// Mitsubishi GX Works2 project: CODE_PLC_HMI   PLC: FX1N/FX1NC

PROGRAM MAIN
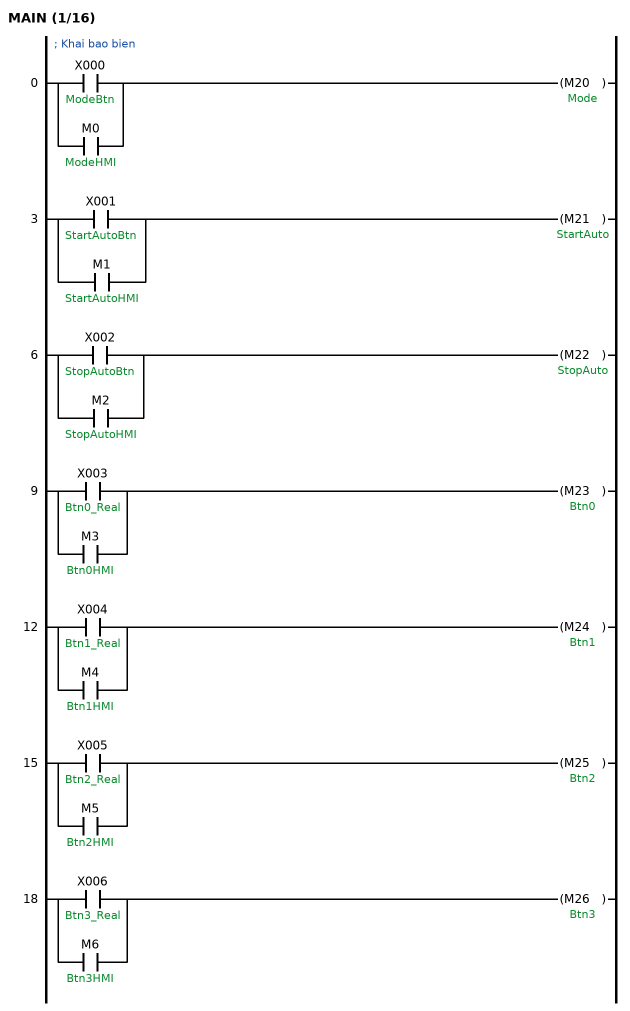
; Khai bao bien
0     LD      X000  ; ModeBtn
      OR      M0  ; ModeHMI
      OUT     M20  ; Mode
3     LD      X001  ; StartAutoBtn
      OR      M1  ; StartAutoHMI
      OUT     M21  ; StartAuto
6     LD      X002  ; StopAutoBtn
      OR      M2  ; StopAutoHMI
      OUT     M22  ; StopAuto
9     LD      X003  ; Btn0_Real
      OR      M3  ; Btn0HMI
      OUT     M23  ; Btn0
12    LD      X004  ; Btn1_Real
      OR      M4  ; Btn1HMI
      OUT     M24  ; Btn1
15    LD      X005  ; Btn2_Real
      OR      M5  ; Btn2HMI
      OUT     M25  ; Btn2
18    LD      X006  ; Btn3_Real
      OR      M6  ; Btn3HMI
      OUT     M26  ; Btn3
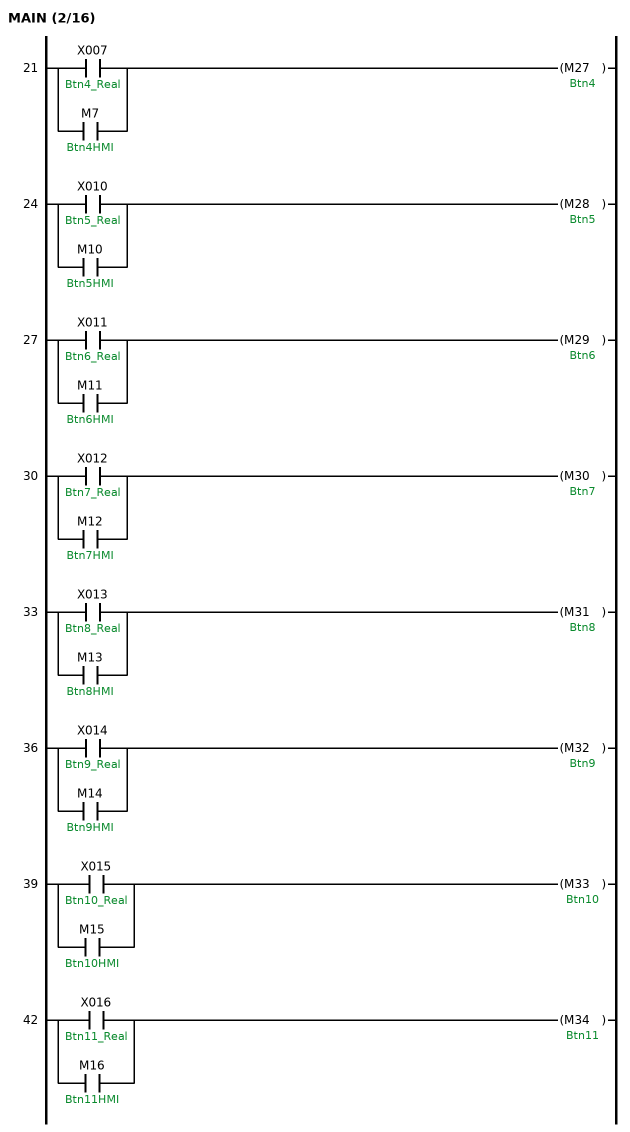
21    LD      X007  ; Btn4_Real
      OR      M7  ; Btn4HMI
      OUT     M27  ; Btn4
24    LD      X010  ; Btn5_Real
      OR      M10  ; Btn5HMI
      OUT     M28  ; Btn5
27    LD      X011  ; Btn6_Real
      OR      M11  ; Btn6HMI
      OUT     M29  ; Btn6
30    LD      X012  ; Btn7_Real
      OR      M12  ; Btn7HMI
      OUT     M30  ; Btn7
33    LD      X013  ; Btn8_Real
      OR      M13  ; Btn8HMI
      OUT     M31  ; Btn8
36    LD      X014  ; Btn9_Real
      OR      M14  ; Btn9HMI
      OUT     M32  ; Btn9
39    LD      X015  ; Btn10_Real
      OR      M15  ; Btn10HMI
      OUT     M33  ; Btn10
42    LD      X016  ; Btn11_Real
      OR      M16  ; Btn11HMI
      OUT     M34  ; Btn11
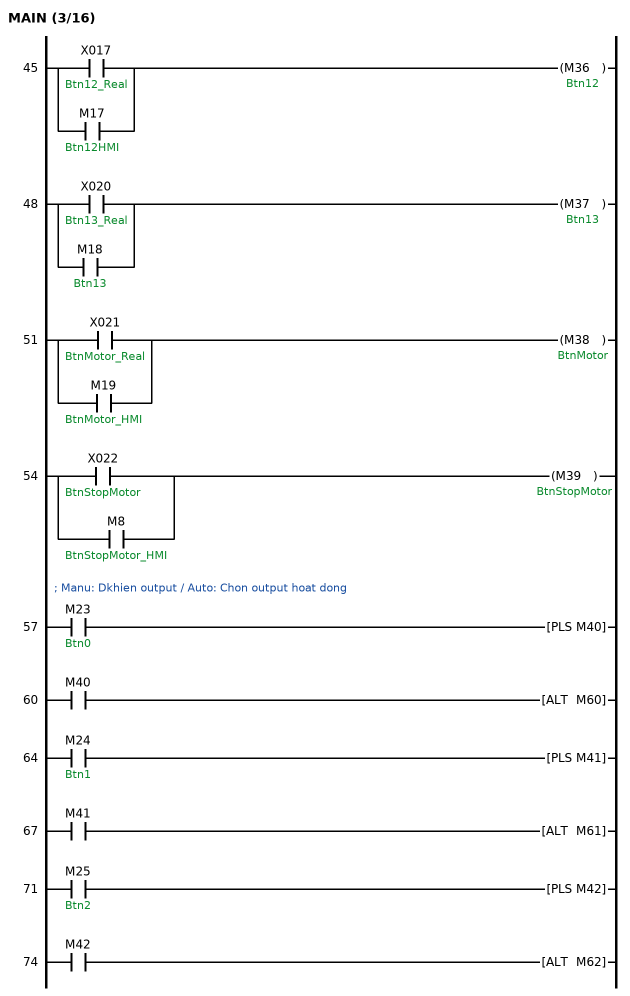
45    LD      X017  ; Btn12_Real
      OR      M17  ; Btn12HMI
      OUT     M36  ; Btn12
48    LD      X020  ; Btn13_Real
      OR      M18  ; Btn13
      OUT     M37  ; Btn13
51    LD      X021  ; BtnMotor_Real
      OR      M19  ; BtnMotor_HMI
      OUT     M38  ; BtnMotor
54    LD      X022  ; BtnStopMotor
      OR      M8  ; BtnStopMotor_HMI
      OUT     M39  ; BtnStopMotor
; Manu: Dkhien output / Auto: Chon output hoat dong
57    LD      M23  ; Btn0
      PLS     M40
60    LD      M40
      ALT     M60
64    LD      M24  ; Btn1
      PLS     M41
67    LD      M41
      ALT     M61
71    LD      M25  ; Btn2
      PLS     M42
74    LD      M42
      ALT     M62
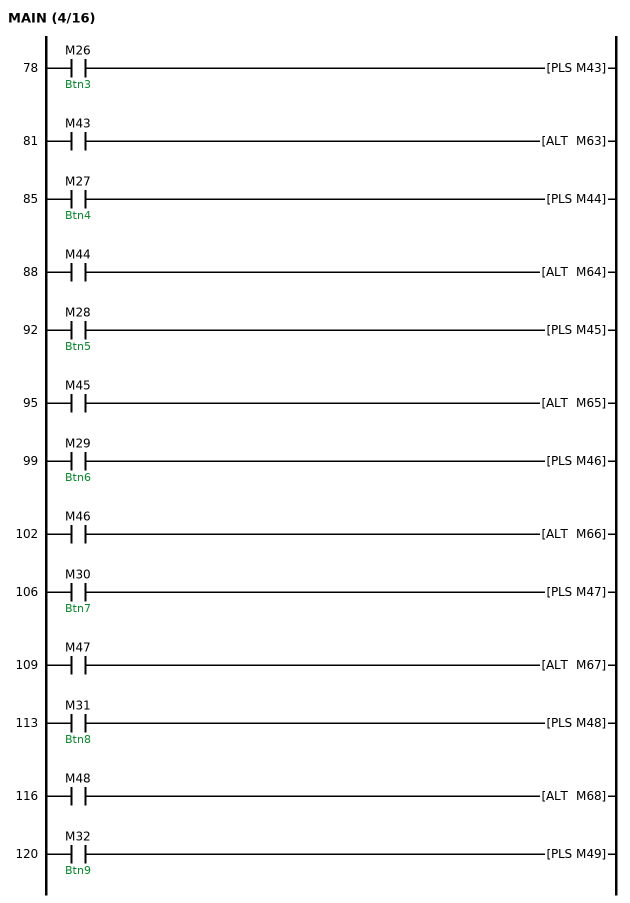
78    LD      M26  ; Btn3
      PLS     M43
81    LD      M43
      ALT     M63
85    LD      M27  ; Btn4
      PLS     M44
88    LD      M44
      ALT     M64
92    LD      M28  ; Btn5
      PLS     M45
95    LD      M45
      ALT     M65
99    LD      M29  ; Btn6
      PLS     M46
102   LD      M46
      ALT     M66
106   LD      M30  ; Btn7
      PLS     M47
109   LD      M47
      ALT     M67
113   LD      M31  ; Btn8
      PLS     M48
116   LD      M48
      ALT     M68
120   LD      M32  ; Btn9
      PLS     M49
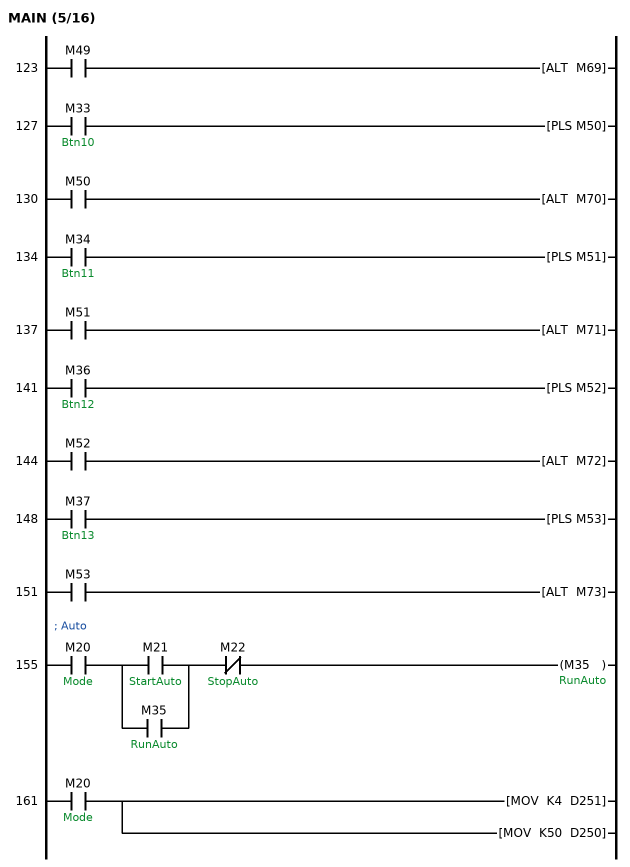
123   LD      M49
      ALT     M69
127   LD      M33  ; Btn10
      PLS     M50
130   LD      M50
      ALT     M70
134   LD      M34  ; Btn11
      PLS     M51
137   LD      M51
      ALT     M71
141   LD      M36  ; Btn12
      PLS     M52
144   LD      M52
      ALT     M72
148   LD      M37  ; Btn13
      PLS     M53
151   LD      M53
      ALT     M73
; 
; Auto
155   LD      M20  ; Mode
      LD      M21  ; StartAuto
      OR      M35  ; RunAuto
      ANB
      ANI     M22  ; StopAuto
      OUT     M35  ; RunAuto
161   LD      M20  ; Mode
      MOV     K4 D251
      MOV     K50 D250
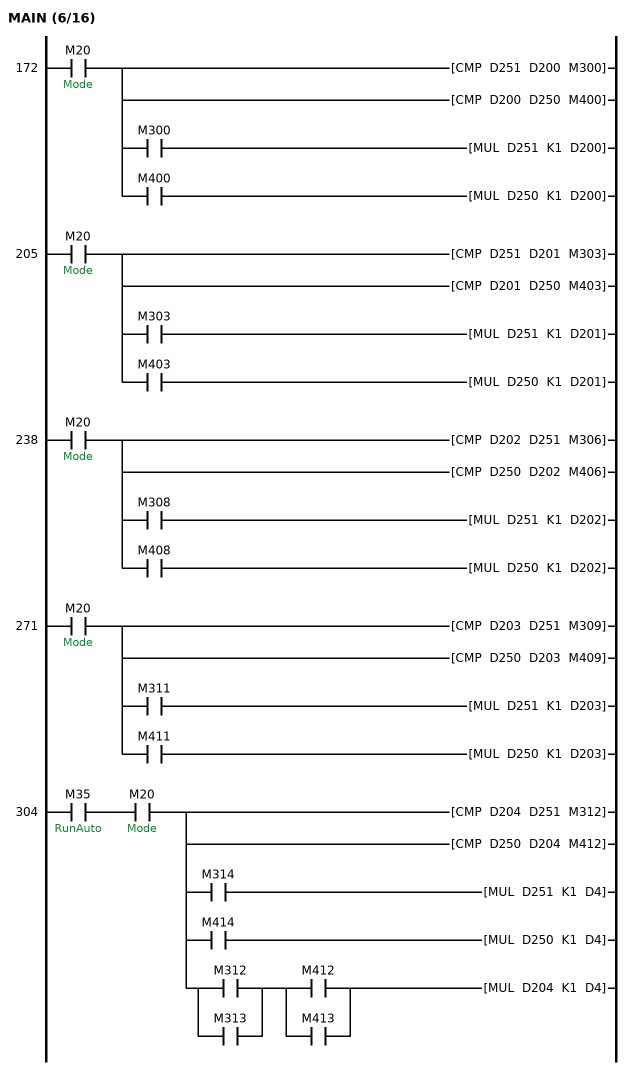
172   LD      M20  ; Mode
      CMP     D251 D200 M300
      CMP     D200 D250 M400
      MPS
      AND     M300
      MUL     D251 K1 D200
      MPP
      AND     M400
      MUL     D250 K1 D200
205   LD      M20  ; Mode
      CMP     D251 D201 M303
      CMP     D201 D250 M403
      MPS
      AND     M303
      MUL     D251 K1 D201
      MPP
      AND     M403
      MUL     D250 K1 D201
238   LD      M20  ; Mode
      CMP     D202 D251 M306
      CMP     D250 D202 M406
      MPS
      AND     M308
      MUL     D251 K1 D202
      MPP
      AND     M408
      MUL     D250 K1 D202
271   LD      M20  ; Mode
      CMP     D203 D251 M309
      CMP     D250 D203 M409
      MPS
      AND     M311
      MUL     D251 K1 D203
      MPP
      AND     M411
      MUL     D250 K1 D203
304   LD      M35  ; RunAuto
      AND     M20  ; Mode
      CMP     D204 D251 M312
      CMP     D250 D204 M412
      MPS
      AND     M314
      MUL     D251 K1 D4
      MRD
      AND     M414
      MUL     D250 K1 D4
      MPP
      LD      M312
      OR      M313
      ANB
      LD      M412
      OR      M413
      ANB
      MUL     D204 K1 D4
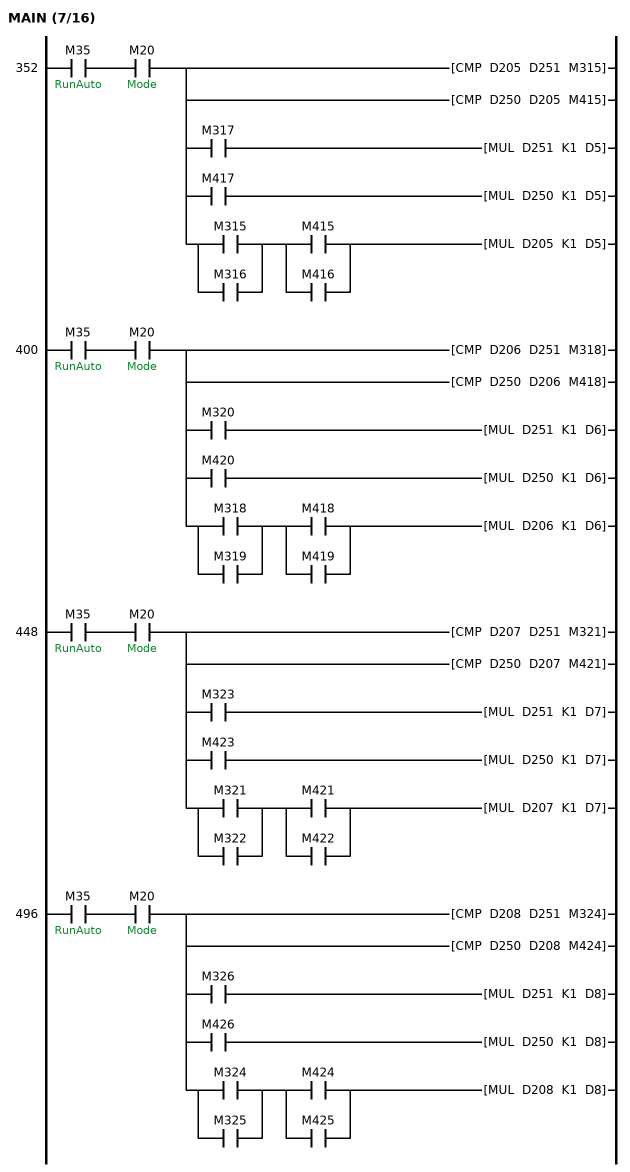
352   LD      M35  ; RunAuto
      AND     M20  ; Mode
      CMP     D205 D251 M315
      CMP     D250 D205 M415
      MPS
      AND     M317
      MUL     D251 K1 D5
      MRD
      AND     M417
      MUL     D250 K1 D5
      MPP
      LD      M315
      OR      M316
      ANB
      LD      M415
      OR      M416
      ANB
      MUL     D205 K1 D5
400   LD      M35  ; RunAuto
      AND     M20  ; Mode
      CMP     D206 D251 M318
      CMP     D250 D206 M418
      MPS
      AND     M320
      MUL     D251 K1 D6
      MRD
      AND     M420
      MUL     D250 K1 D6
      MPP
      LD      M318
      OR      M319
      ANB
      LD      M418
      OR      M419
      ANB
      MUL     D206 K1 D6
448   LD      M35  ; RunAuto
      AND     M20  ; Mode
      CMP     D207 D251 M321
      CMP     D250 D207 M421
      MPS
      AND     M323
      MUL     D251 K1 D7
      MRD
      AND     M423
      MUL     D250 K1 D7
      MPP
      LD      M321
      OR      M322
      ANB
      LD      M421
      OR      M422
      ANB
      MUL     D207 K1 D7
496   LD      M35  ; RunAuto
      AND     M20  ; Mode
      CMP     D208 D251 M324
      CMP     D250 D208 M424
      MPS
      AND     M326
      MUL     D251 K1 D8
      MRD
      AND     M426
      MUL     D250 K1 D8
      MPP
      LD      M324
      OR      M325
      ANB
      LD      M424
      OR      M425
      ANB
      MUL     D208 K1 D8
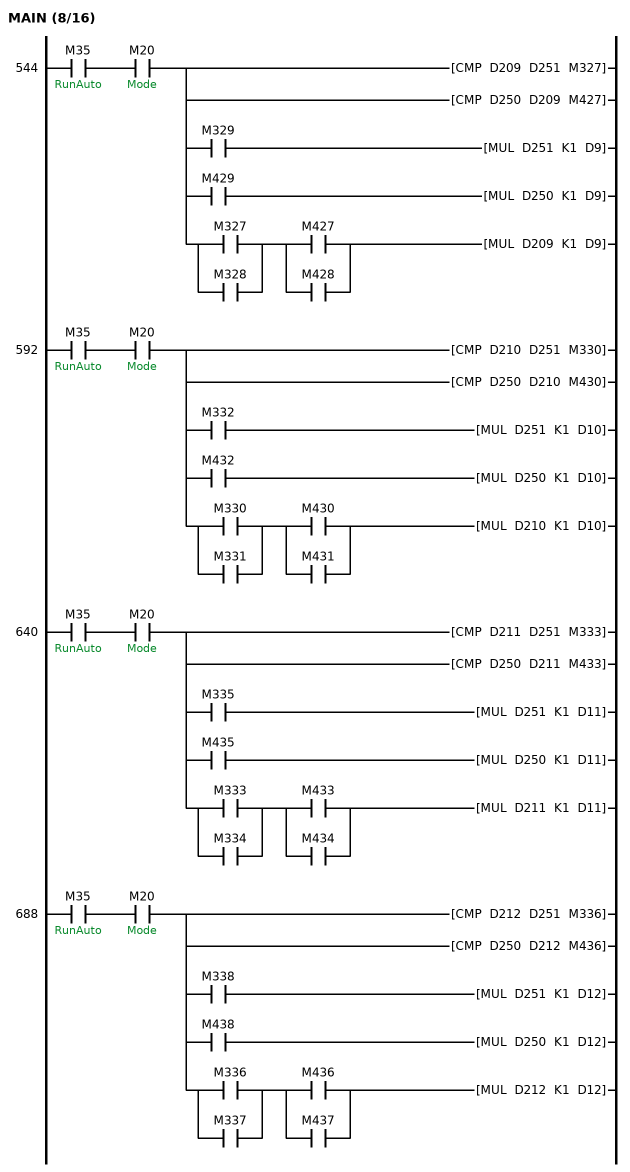
544   LD      M35  ; RunAuto
      AND     M20  ; Mode
      CMP     D209 D251 M327
      CMP     D250 D209 M427
      MPS
      AND     M329
      MUL     D251 K1 D9
      MRD
      AND     M429
      MUL     D250 K1 D9
      MPP
      LD      M327
      OR      M328
      ANB
      LD      M427
      OR      M428
      ANB
      MUL     D209 K1 D9
592   LD      M35  ; RunAuto
      AND     M20  ; Mode
      CMP     D210 D251 M330
      CMP     D250 D210 M430
      MPS
      AND     M332
      MUL     D251 K1 D10
      MRD
      AND     M432
      MUL     D250 K1 D10
      MPP
      LD      M330
      OR      M331
      ANB
      LD      M430
      OR      M431
      ANB
      MUL     D210 K1 D10
640   LD      M35  ; RunAuto
      AND     M20  ; Mode
      CMP     D211 D251 M333
      CMP     D250 D211 M433
      MPS
      AND     M335
      MUL     D251 K1 D11
      MRD
      AND     M435
      MUL     D250 K1 D11
      MPP
      LD      M333
      OR      M334
      ANB
      LD      M433
      OR      M434
      ANB
      MUL     D211 K1 D11
688   LD      M35  ; RunAuto
      AND     M20  ; Mode
      CMP     D212 D251 M336
      CMP     D250 D212 M436
      MPS
      AND     M338
      MUL     D251 K1 D12
      MRD
      AND     M438
      MUL     D250 K1 D12
      MPP
      LD      M336
      OR      M337
      ANB
      LD      M436
      OR      M437
      ANB
      MUL     D212 K1 D12
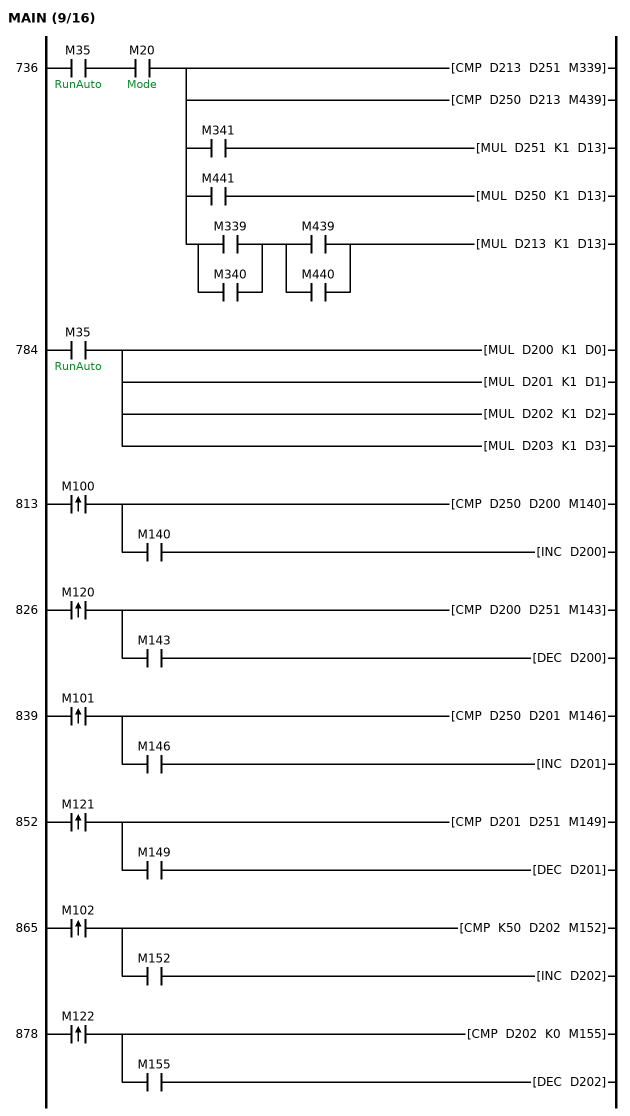
736   LD      M35  ; RunAuto
      AND     M20  ; Mode
      CMP     D213 D251 M339
      CMP     D250 D213 M439
      MPS
      AND     M341
      MUL     D251 K1 D13
      MRD
      AND     M441
      MUL     D250 K1 D13
      MPP
      LD      M339
      OR      M340
      ANB
      LD      M439
      OR      M440
      ANB
      MUL     D213 K1 D13
784   LD      M35  ; RunAuto
      MUL     D200 K1 D0
      MUL     D201 K1 D1
      MUL     D202 K1 D2
      MUL     D203 K1 D3
813   LDP     M100
      CMP     D250 D200 M140
      AND     M140
      INC     D200
826   LDP     M120
      CMP     D200 D251 M143
      AND     M143
      DEC     D200
839   LDP     M101
      CMP     D250 D201 M146
      AND     M146
      INC     D201
852   LDP     M121
      CMP     D201 D251 M149
      AND     M149
      DEC     D201
865   LDP     M102
      CMP     K50 D202 M152
      AND     M152
      INC     D202
878   LDP     M122
      CMP     D202 K0 M155
      AND     M155
      DEC     D202
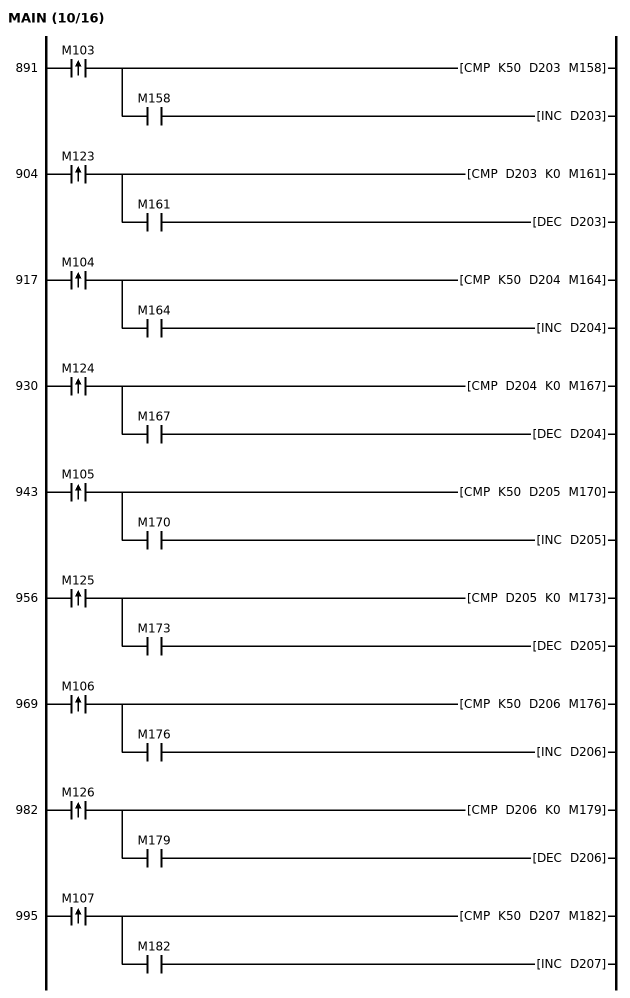
891   LDP     M103
      CMP     K50 D203 M158
      AND     M158
      INC     D203
904   LDP     M123
      CMP     D203 K0 M161
      AND     M161
      DEC     D203
917   LDP     M104
      CMP     K50 D204 M164
      AND     M164
      INC     D204
930   LDP     M124
      CMP     D204 K0 M167
      AND     M167
      DEC     D204
943   LDP     M105
      CMP     K50 D205 M170
      AND     M170
      INC     D205
956   LDP     M125
      CMP     D205 K0 M173
      AND     M173
      DEC     D205
969   LDP     M106
      CMP     K50 D206 M176
      AND     M176
      INC     D206
982   LDP     M126
      CMP     D206 K0 M179
      AND     M179
      DEC     D206
995   LDP     M107
      CMP     K50 D207 M182
      AND     M182
      INC     D207
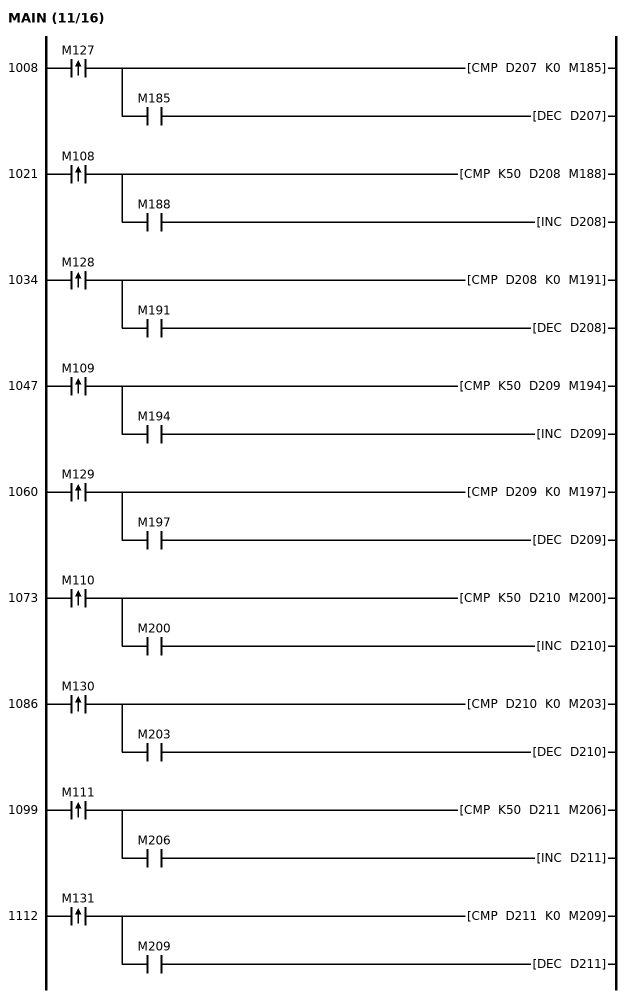
1008  LDP     M127
      CMP     D207 K0 M185
      AND     M185
      DEC     D207
1021  LDP     M108
      CMP     K50 D208 M188
      AND     M188
      INC     D208
1034  LDP     M128
      CMP     D208 K0 M191
      AND     M191
      DEC     D208
1047  LDP     M109
      CMP     K50 D209 M194
      AND     M194
      INC     D209
1060  LDP     M129
      CMP     D209 K0 M197
      AND     M197
      DEC     D209
1073  LDP     M110
      CMP     K50 D210 M200
      AND     M200
      INC     D210
1086  LDP     M130
      CMP     D210 K0 M203
      AND     M203
      DEC     D210
1099  LDP     M111
      CMP     K50 D211 M206
      AND     M206
      INC     D211
1112  LDP     M131
      CMP     D211 K0 M209
      AND     M209
      DEC     D211
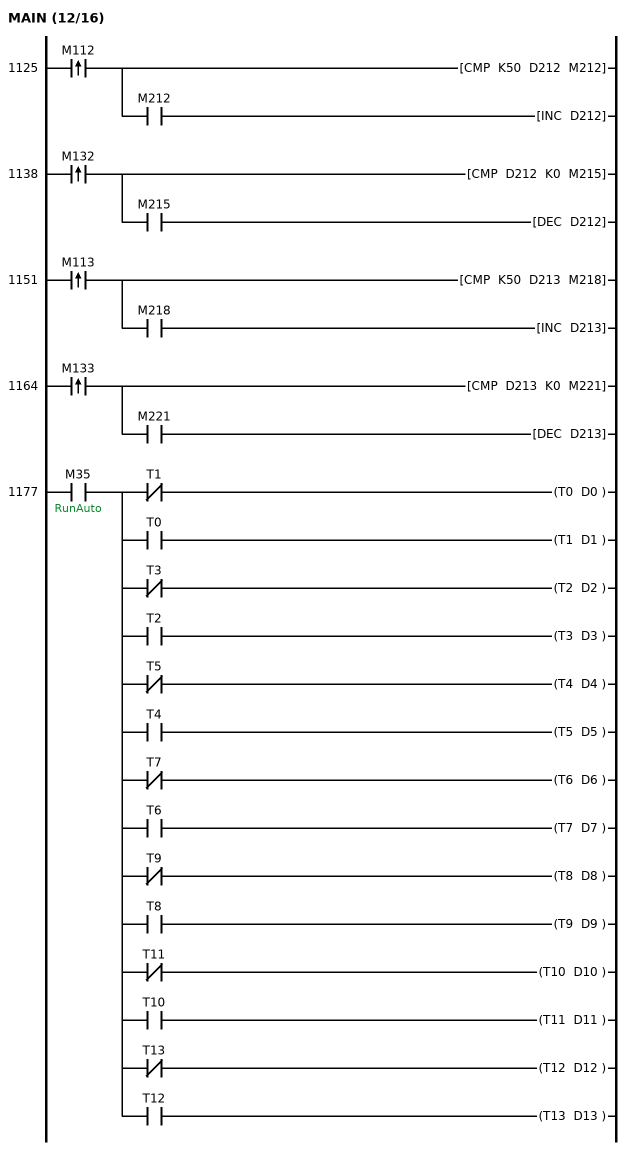
1125  LDP     M112
      CMP     K50 D212 M212
      AND     M212
      INC     D212
1138  LDP     M132
      CMP     D212 K0 M215
      AND     M215
      DEC     D212
1151  LDP     M113
      CMP     K50 D213 M218
      AND     M218
      INC     D213
1164  LDP     M133
      CMP     D213 K0 M221
      AND     M221
      DEC     D213
1177  LD      M35  ; RunAuto
      MPS
      ANI     T1
      OUT     T0 D0
      MRD
      AND     T0
      OUT     T1 D1
      MRD
      ANI     T3
      OUT     T2 D2
      MRD
      AND     T2
      OUT     T3 D3
      MRD
      ANI     T5
      OUT     T4 D4
      MRD
      AND     T4
      OUT     T5 D5
      MRD
      ANI     T7
      OUT     T6 D6
      MRD
      AND     T6
      OUT     T7 D7
      MRD
      ANI     T9
      OUT     T8 D8
      MRD
      AND     T8
      OUT     T9 D9
      MRD
      ANI     T11
      OUT     T10 D10
      MRD
      AND     T10
      OUT     T11 D11
      MRD
      ANI     T13
      OUT     T12 D12
      MPP
      AND     T12
      OUT     T13 D13
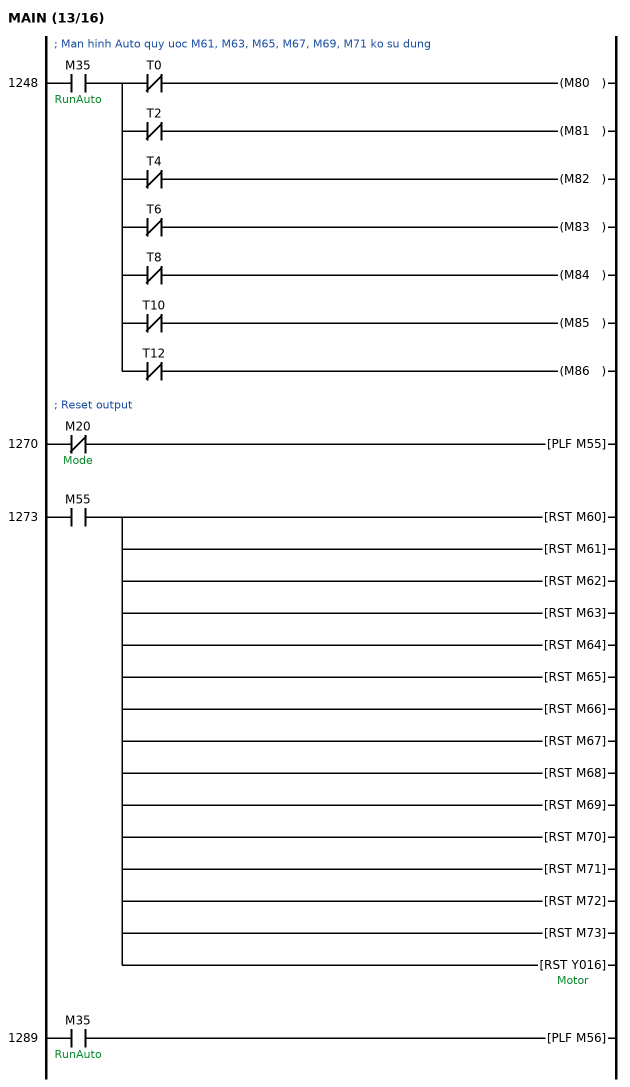
; Man hinh Auto quy uoc M61, M63, M65, M67, M69, M71 ko su dung
1248  LD      M35  ; RunAuto
      MPS
      ANI     T0
      OUT     M80
      MRD
      ANI     T2
      OUT     M81
      MRD
      ANI     T4
      OUT     M82
      MRD
      ANI     T6
      OUT     M83
      MRD
      ANI     T8
      OUT     M84
      MRD
      ANI     T10
      OUT     M85
      MPP
      ANI     T12
      OUT     M86
; 
; Reset output
1270  LDI     M20  ; Mode
      PLF     M55
1273  LD      M55
      RST     M60
      RST     M61
      RST     M62
      RST     M63
      RST     M64
      RST     M65
      RST     M66
      RST     M67
      RST     M68
      RST     M69
      RST     M70
      RST     M71
      RST     M72
      RST     M73
      RST     Y016  ; Motor
1289  LD      M35  ; RunAuto
      PLF     M56
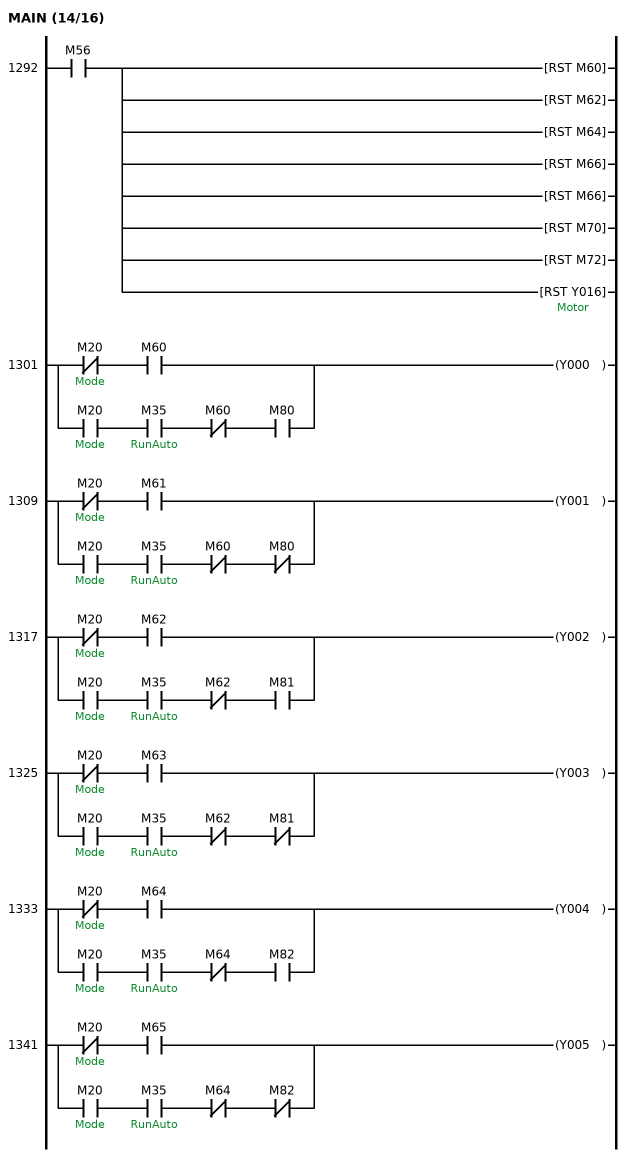
1292  LD      M56
      RST     M60
      RST     M62
      RST     M64
      RST     M66
      RST     M66
      RST     M70
      RST     M72
      RST     Y016  ; Motor
1301  LDI     M20  ; Mode
      AND     M60
      LD      M20  ; Mode
      AND     M35  ; RunAuto
      ANI     M60
      AND     M80
      ORB
      OUT     Y000
1309  LDI     M20  ; Mode
      AND     M61
      LD      M20  ; Mode
      AND     M35  ; RunAuto
      ANI     M60
      ANI     M80
      ORB
      OUT     Y001
1317  LDI     M20  ; Mode
      AND     M62
      LD      M20  ; Mode
      AND     M35  ; RunAuto
      ANI     M62
      AND     M81
      ORB
      OUT     Y002
1325  LDI     M20  ; Mode
      AND     M63
      LD      M20  ; Mode
      AND     M35  ; RunAuto
      ANI     M62
      ANI     M81
      ORB
      OUT     Y003
1333  LDI     M20  ; Mode
      AND     M64
      LD      M20  ; Mode
      AND     M35  ; RunAuto
      ANI     M64
      AND     M82
      ORB
      OUT     Y004
1341  LDI     M20  ; Mode
      AND     M65
      LD      M20  ; Mode
      AND     M35  ; RunAuto
      ANI     M64
      ANI     M82
      ORB
      OUT     Y005
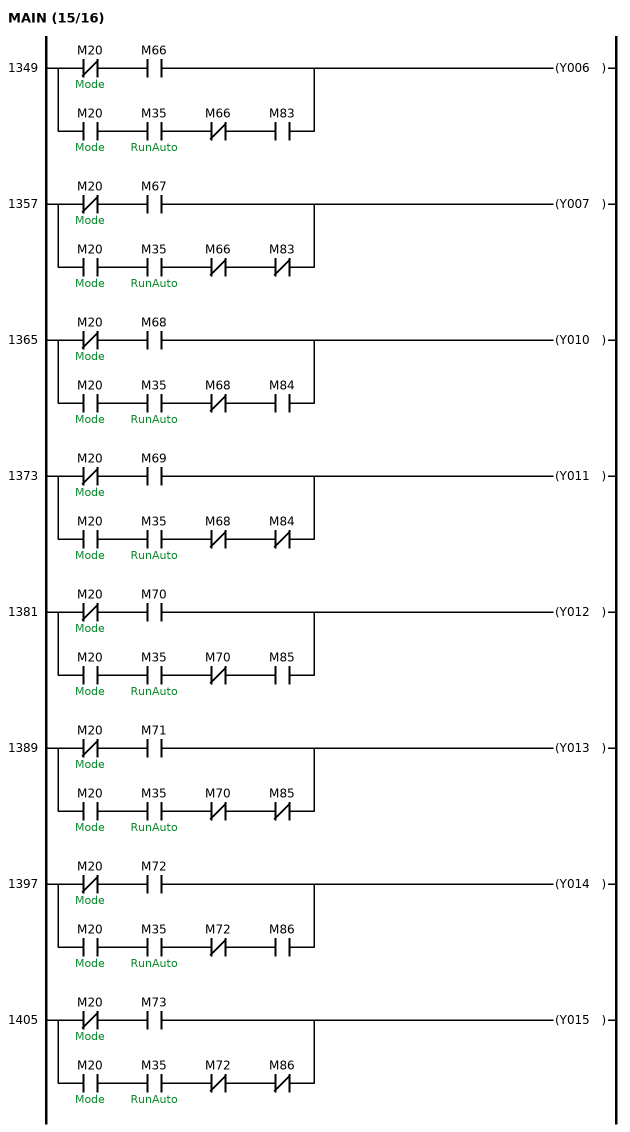
1349  LDI     M20  ; Mode
      AND     M66
      LD      M20  ; Mode
      AND     M35  ; RunAuto
      ANI     M66
      AND     M83
      ORB
      OUT     Y006
1357  LDI     M20  ; Mode
      AND     M67
      LD      M20  ; Mode
      AND     M35  ; RunAuto
      ANI     M66
      ANI     M83
      ORB
      OUT     Y007
1365  LDI     M20  ; Mode
      AND     M68
      LD      M20  ; Mode
      AND     M35  ; RunAuto
      ANI     M68
      AND     M84
      ORB
      OUT     Y010
1373  LDI     M20  ; Mode
      AND     M69
      LD      M20  ; Mode
      AND     M35  ; RunAuto
      ANI     M68
      ANI     M84
      ORB
      OUT     Y011
1381  LDI     M20  ; Mode
      AND     M70
      LD      M20  ; Mode
      AND     M35  ; RunAuto
      ANI     M70
      AND     M85
      ORB
      OUT     Y012
1389  LDI     M20  ; Mode
      AND     M71
      LD      M20  ; Mode
      AND     M35  ; RunAuto
      ANI     M70
      ANI     M85
      ORB
      OUT     Y013
1397  LDI     M20  ; Mode
      AND     M72
      LD      M20  ; Mode
      AND     M35  ; RunAuto
      ANI     M72
      AND     M86
      ORB
      OUT     Y014
1405  LDI     M20  ; Mode
      AND     M73
      LD      M20  ; Mode
      AND     M35  ; RunAuto
      ANI     M72
      ANI     M86
      ORB
      OUT     Y015
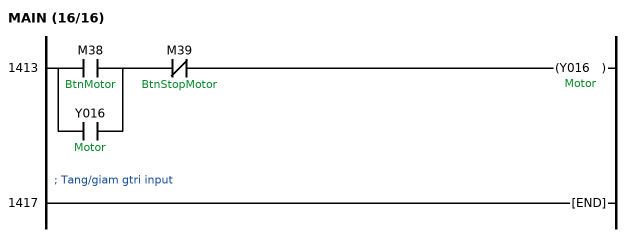
1413  LD      M38  ; BtnMotor
      OR      Y016  ; Motor
      ANI     M39  ; BtnStopMotor
      OUT     Y016  ; Motor
; Tang/giam gtri input
1417  END
END_PROGRAM
